(* CODESYS project GitTest
   Author: SESA103994
   Title: Untitled450
   Version: 0.0.0.0

Project tree, tasks and I/O mapping:
  LMC_PacDrive : PacDrive LMC 300/400/402/600/802/902C, Schneider Electric, order no. LMC Pro and Pro2, version 1.76.14.2
    application Application
      task TASK_SR_Main (cyclic, interval t#10ms, priority 14, watchdog 100 ms x 10) calls SR_Main
      program SR_Main [ST]
    Device Addressing
    Message Logger
    AI_0 : Analog Input, Schneider Electric, version 1.76.14.2
    AI_1 : Analog Input, Schneider Electric, version 1.76.14.2
    AQ_0 : Analog Output, Schneider Electric, version 1.76.14.2
    AQ_1 : Analog Output, Schneider Electric, version 1.76.14.2
    DIG_DigitalIn : Digital Inputs, Schneider Electric, version 1.76.14.2
      DI_0 : Input, Schneider Electric, version 1.76.14.2
      DI_10 : Input, Schneider Electric, version 1.76.14.2
      DI_11 : Input, Schneider Electric, version 1.76.14.2
      DI_12 : Input, Schneider Electric, version 1.76.14.2
      DI_13 : Input, Schneider Electric, version 1.76.14.2
      DI_14 : Input, Schneider Electric, version 1.76.14.2
      DI_15 : Input, Schneider Electric, version 1.76.14.2
      DI_16 : Input, Schneider Electric, version 1.76.14.2
      DI_17 : Input, Schneider Electric, version 1.76.14.2
      DI_18 : Input, Schneider Electric, version 1.76.14.2
      DI_19 : Input, Schneider Electric, version 1.76.14.2
      DI_1 : Input, Schneider Electric, version 1.76.14.2
      DI_2 : Input, Schneider Electric, version 1.76.14.2
      DI_3 : Input, Schneider Electric, version 1.76.14.2
      DI_4 : Input, Schneider Electric, version 1.76.14.2
      DI_5 : Input, Schneider Electric, version 1.76.14.2
      DI_6 : Input, Schneider Electric, version 1.76.14.2
      DI_7 : Input, Schneider Electric, version 1.76.14.2
      DI_8 : Input, Schneider Electric, version 1.76.14.2
      DI_9 : Input, Schneider Electric, version 1.76.14.2
      FI_0 : Fast Input, Schneider Electric, version 1.76.14.2
      FI_1 : Fast Input, Schneider Electric, version 1.76.14.2
      FI_2 : Fast Input, Schneider Electric, version 1.76.14.2
      FI_3 : Fast Input, Schneider Electric, version 1.76.14.2
    DQG_DigitalOut : Digital Outputs, Schneider Electric, version 1.76.14.2
      DQ_0 : Output, Schneider Electric, version 1.76.14.2
      DQ_10 : Output, Schneider Electric, version 1.76.14.2
      DQ_11 : Output, Schneider Electric, version 1.76.14.2
      DQ_12 : Output, Schneider Electric, version 1.76.14.2
      DQ_13 : Output, Schneider Electric, version 1.76.14.2
      DQ_14 : Output, Schneider Electric, version 1.76.14.2
      DQ_15 : Output, Schneider Electric, version 1.76.14.2
      DQ_1 : Output, Schneider Electric, version 1.76.14.2
      DQ_2 : Output, Schneider Electric, version 1.76.14.2
      DQ_3 : Output, Schneider Electric, version 1.76.14.2
      DQ_4 : Output, Schneider Electric, version 1.76.14.2
      DQ_5 : Output, Schneider Electric, version 1.76.14.2
      DQ_6 : Output, Schneider Electric, version 1.76.14.2
      DQ_7 : Output, Schneider Electric, version 1.76.14.2
      DQ_8 : Output, Schneider Electric, version 1.76.14.2
      DQ_9 : Output, Schneider Electric, version 1.76.14.2
    Sercos_Master : Sercos Master, Schneider Electric, version 1.76.14.2
    TPG_TPIn : Touch Probe Inputs, Schneider Electric, version 1.76.14.2
      TP_0 : Touch Probe Input, Schneider Electric, version 1.76.14.2
      TP_10 : Touch Probe Input, Schneider Electric, version 1.76.14.2
      TP_11 : Touch Probe Input, Schneider Electric, version 1.76.14.2
      TP_12 : Touch Probe Input, Schneider Electric, version 1.76.14.2
      TP_13 : Touch Probe Input, Schneider Electric, version 1.76.14.2
      TP_14 : Touch Probe Input, Schneider Electric, version 1.76.14.2
      TP_15 : Touch Probe Input, Schneider Electric, version 1.76.14.2
      TP_1 : Touch Probe Input, Schneider Electric, version 1.76.14.2
      TP_2 : Touch Probe Input, Schneider Electric, version 1.76.14.2
      TP_3 : Touch Probe Input, Schneider Electric, version 1.76.14.2
      TP_4 : Touch Probe Input, Schneider Electric, version 1.76.14.2
      TP_5 : Touch Probe Input, Schneider Electric, version 1.76.14.2
      TP_6 : Touch Probe Input, Schneider Electric, version 1.76.14.2
      TP_7 : Touch Probe Input, Schneider Electric, version 1.76.14.2
      TP_8 : Touch Probe Input, Schneider Electric, version 1.76.14.2
      TP_9 : Touch Probe Input, Schneider Electric, version 1.76.14.2
  LMC_PacDrive : PacDrive LMC 300/400/402/600/802/902C, Schneider Electric, order no. LMC Pro and Pro2, version 1.76.14.2
    application Application
      task TASK_SR_Main (cyclic, interval t#10ms, priority 14, watchdog 100 ms x 10) calls SR_Main
      program SR_Main [ST]
    Device Addressing
    Message Logger
    AI_0 : Analog Input, Schneider Electric, version 1.76.14.2
    AI_1 : Analog Input, Schneider Electric, version 1.76.14.2
    AQ_0 : Analog Output, Schneider Electric, version 1.76.14.2
    AQ_1 : Analog Output, Schneider Electric, version 1.76.14.2
    DIG_DigitalIn : Digital Inputs, Schneider Electric, version 1.76.14.2
      DI_0 : Input, Schneider Electric, version 1.76.14.2
      DI_10 : Input, Schneider Electric, version 1.76.14.2
      DI_11 : Input, Schneider Electric, version 1.76.14.2
      DI_12 : Input, Schneider Electric, version 1.76.14.2
      DI_13 : Input, Schneider Electric, version 1.76.14.2
      DI_14 : Input, Schneider Electric, version 1.76.14.2
      DI_15 : Input, Schneider Electric, version 1.76.14.2
      DI_16 : Input, Schneider Electric, version 1.76.14.2
      DI_17 : Input, Schneider Electric, version 1.76.14.2
      DI_18 : Input, Schneider Electric, version 1.76.14.2
      DI_19 : Input, Schneider Electric, version 1.76.14.2
      DI_1 : Input, Schneider Electric, version 1.76.14.2
      DI_2 : Input, Schneider Electric, version 1.76.14.2
      DI_3 : Input, Schneider Electric, version 1.76.14.2
      DI_4 : Input, Schneider Electric, version 1.76.14.2
      DI_5 : Input, Schneider Electric, version 1.76.14.2
      DI_6 : Input, Schneider Electric, version 1.76.14.2
      DI_7 : Input, Schneider Electric, version 1.76.14.2
      DI_8 : Input, Schneider Electric, version 1.76.14.2
      DI_9 : Input, Schneider Electric, version 1.76.14.2
      FI_0 : Fast Input, Schneider Electric, version 1.76.14.2
      FI_1 : Fast Input, Schneider Electric, version 1.76.14.2
      FI_2 : Fast Input, Schneider Electric, version 1.76.14.2
      FI_3 : Fast Input, Schneider Electric, version 1.76.14.2
    DQG_DigitalOut : Digital Outputs, Schneider Electric, version 1.76.14.2
      DQ_0 : Output, Schneider Electric, version 1.76.14.2
      DQ_10 : Output, Schneider Electric, version 1.76.14.2
      DQ_11 : Output, Schneider Electric, version 1.76.14.2
      DQ_12 : Output, Schneider Electric, version 1.76.14.2
      DQ_13 : Output, Schneider Electric, version 1.76.14.2
      DQ_14 : Output, Schneider Electric, version 1.76.14.2
      DQ_15 : Output, Schneider Electric, version 1.76.14.2
      DQ_1 : Output, Schneider Electric, version 1.76.14.2
      DQ_2 : Output, Schneider Electric, version 1.76.14.2
      DQ_3 : Output, Schneider Electric, version 1.76.14.2
      DQ_4 : Output, Schneider Electric, version 1.76.14.2
      DQ_5 : Output, Schneider Electric, version 1.76.14.2
      DQ_6 : Output, Schneider Electric, version 1.76.14.2
      DQ_7 : Output, Schneider Electric, version 1.76.14.2
      DQ_8 : Output, Schneider Electric, version 1.76.14.2
      DQ_9 : Output, Schneider Electric, version 1.76.14.2
    Sercos_Master : Sercos Master, Schneider Electric, version 1.76.14.2
    TPG_TPIn : Touch Probe Inputs, Schneider Electric, version 1.76.14.2
      TP_0 : Touch Probe Input, Schneider Electric, version 1.76.14.2
      TP_10 : Touch Probe Input, Schneider Electric, version 1.76.14.2
      TP_11 : Touch Probe Input, Schneider Electric, version 1.76.14.2
      TP_12 : Touch Probe Input, Schneider Electric, version 1.76.14.2
      TP_13 : Touch Probe Input, Schneider Electric, version 1.76.14.2
      TP_14 : Touch Probe Input, Schneider Electric, version 1.76.14.2
      TP_15 : Touch Probe Input, Schneider Electric, version 1.76.14.2
      TP_1 : Touch Probe Input, Schneider Electric, version 1.76.14.2
      TP_2 : Touch Probe Input, Schneider Electric, version 1.76.14.2
      TP_3 : Touch Probe Input, Schneider Electric, version 1.76.14.2
      TP_4 : Touch Probe Input, Schneider Electric, version 1.76.14.2
      TP_5 : Touch Probe Input, Schneider Electric, version 1.76.14.2
      TP_6 : Touch Probe Input, Schneider Electric, version 1.76.14.2
      TP_7 : Touch Probe Input, Schneider Electric, version 1.76.14.2
      TP_8 : Touch Probe Input, Schneider Electric, version 1.76.14.2
      TP_9 : Touch Probe Input, Schneider Electric, version 1.76.14.2
  function GetTextProperty2 [ST]
  function GetTextProperty [ST]
  function GetTitle [ST]
  function GetVersionProperty [ST]
*)

// LMC_PacDrive/Application/SR_Main
PROGRAM SR_Main
VAR
END_VAR

END_PROGRAM

// LMC_PacDrive/Application/SR_Main
PROGRAM SR_Main
VAR
END_VAR

END_PROGRAM

// GetTextProperty2
// This function has been automatically generated from the project information.
{attribute 'signature_flag' := '1073741824'}
{attribute 'register_in_runtime'}
FUNCTION GetTextProperty2 : POINTER TO WSTRING
VAR_INPUT
	stKey: WSTRING;
END_VAR

IF stKey = "Author" THEN
	GetTextProperty2 := ADR("SESA103994");
ELSIF stKey = "Company" THEN
	GetTextProperty2 := ADR("");
ELSIF stKey = "Description" THEN
	GetTextProperty2 := ADR("");
ELSIF stKey = "Project" THEN
	GetTextProperty2 := ADR("Untitled450");
ELSIF stKey = "Title" THEN
	GetTextProperty2 := ADR("Untitled450");
ELSE
	GetTextProperty2 := ADR("");
END_IF

END_FUNCTION

// GetTextProperty
// This function has been automatically generated from the project information.
{attribute 'signature_flag' := '1073741824'}
{attribute 'register_in_runtime'}
FUNCTION GetTextProperty : WSTRING
VAR_INPUT
	stKey: WSTRING;
END_VAR

IF stKey = "Author" THEN
	GetTextProperty := "SESA103994";
ELSIF stKey = "Company" THEN
	GetTextProperty := "";
ELSIF stKey = "Description" THEN
	GetTextProperty := "";
ELSIF stKey = "Project" THEN
	GetTextProperty := "Untitled450";
ELSIF stKey = "Title" THEN
	GetTextProperty := "Untitled450";
ELSE
	GetTextProperty := "";
END_IF

END_FUNCTION

// GetTitle
// This function has been automatically generated from the project information.
{attribute 'signature_flag' := '1073741824'}
{attribute 'register_in_runtime'}
FUNCTION GetTitle : WSTRING
VAR_INPUT
	
END_VAR

GetTitle := "Untitled450";

END_FUNCTION

// GetVersionProperty
// This function has been automatically generated from the project information.
{attribute 'signature_flag' := '1073741824'}
{attribute 'register_in_runtime'}
FUNCTION GetVersionProperty : VERSION
VAR_INPUT
	stKey: WSTRING;
END_VAR

IF stKey = "Version" THEN
	GetVersionProperty.uiMajor := 0;
	GetVersionProperty.uiMinor := 0;
	GetVersionProperty.uiServicePack := 0;
	GetVersionProperty.uiPatch := 0;
ELSE
	GetVersionProperty.uiMajor := 0;
	GetVersionProperty.uiMinor := 0;
	GetVersionProperty.uiServicePack := 0;
	GetVersionProperty.uiPatch := 0;
END_IF

END_FUNCTION
